(*********************************** G.D S.p.A. - Technical Department ***********************************
============= PROGRAM INFO ============
FOLDER:             TBD
MACHINES INVOLVED:  TBD 

============= DESCRIPTION =============
csp machine declaration

============= REVISIONS ===============
Date		Version	 	Author      	Description             
----------	-------		------------  	--------------------------------------------
2019/04/05 	0000.00	 	M.Grasso		Creation of the PRG

**********************************************************************************************************)
(*$R process_ref := prc; $*)
PROGRAM csp_case_feed_shuttle_sensors_ls
VAR
	
	prc:											process;
	prc_path:										STRING;
	
	part_present_di:								digital_input;

END_VAR

_read_var_input();

_object_manager();

IF NOT objects_running()
THEN
	RETURN;	
END_IF

_read_process_image();

_mode_manager();

_set_runtime_properties();

(********************************* BODY *********************************)
(************************************************************************)

_handle_messages();

_write_output();

ACTION _handle_messages:
;
END_ACTION

ACTION _handle_process_test:
;
END_ACTION

ACTION _mode_manager:
IF process_mode_req_is_pending(prc)
THEN
    process_apply_mode_req_first_step(prc);
    CASE process_get_mode(prc) OF
        MODE_TO_ABSENT:
			;
        MODE_TO_INACTIVE:
			;
        MODE_TO_TEST:
			;
        MODE_TO_OPERATIONAL:
			;
    END_CASE
    process_apply_mode_req_second_step(prc);
END_IF
END_ACTION

ACTION _object_manager:
IF objects_initialization()
THEN
	sub_process_init(
		object_name					:= 'csp_case_feed_shuttle_sensors_ls.prc', 
		process						:= csp_case_feed_shuttle_sensors.prc, 
		CONVERSION_this				:= prc);
		
	prc_path 						:= process_get_path(prc);
	
	digital_input_init(
		object_name					:= CONCAT(prc_path, '_part_present_di'), 
		polarity_direct				:= TRUE, 
		process						:= prc, 
		CONVERSION_this				:= part_present_di);
	
	
END_IF

IF objects_running()
THEN
	process_cycle(prc);
END_IF
END_ACTION

ACTION _read_process_image:
;
END_ACTION

ACTION _read_var_input:
;
END_ACTION

ACTION _set_runtime_properties:
;
END_ACTION

ACTION _write_output:
;
END_ACTION

END_PROGRAM

(* stored: Version 1.1.0.1, ProductVersion 3.1.4024.3
   POU csp_case_feed_shuttle_sensors_ls: Id {0e8b88cd-7fd8-4b02-8b56-5ec8ad5ffb84}, SpecialFunc None
   Action _handle_messages: Id {8735e19c-a6e7-4a45-b900-9975544828b6}
   Action _handle_process_test: Id {b42935df-0469-45e1-b72a-bcd7ad78391f}
   Action _mode_manager: Id {123e4798-d861-4426-a539-ae71e32b5b1d}
   Action _object_manager: Id {8871e1e8-cb5e-4e13-a5e5-eec0fcefcc70}
   Action _read_process_image: Id {9a4c75b1-e54d-4d6f-87cb-162baf664b50}
   Action _read_var_input: Id {67fc88b3-77d0-43a8-b59e-458048b8f4bd}
   Action _set_runtime_properties: Id {470bb888-80bd-4bb3-92f2-06df2fccff5c}
   Action _write_output: Id {d0efc4c0-438c-4778-b6ef-b3db703f82db} *)
